Yaskawa INFORM job: BATMAN_ALL2.JBI

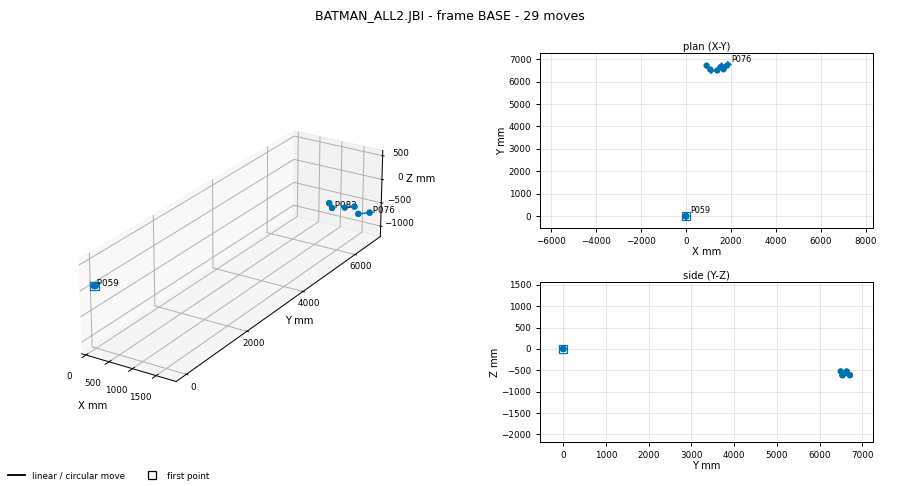
[picture p0: tool path of BATMAN_ALL2.JBI in frame BASE, 29 of 158 moves have a stored position in this frame; points joined in program order, loops and branches not executed]
/JOB
//NAME BATMAN_ALL2
///FOLDERNAME KRIS-SCIANA
//POS
///NPOS 87,87,0,38,0,0
///TOOL 0
///POSTYPE PULSE
///PULSE
C00000=110506,-37041,-50550,-2931,89884,-21361
C00001=114892,-14127,-29600,-10669,91134,-4857
C00002=113309,1036,-13095,-10480,88604,-5183
C00003=113309,1047,-12858,-10479,88468,-5172
C00004=113309,1099,-12019,-10480,87986,-5131
C00005=110003,-19213,-30454,-10104,88460,-6296
C00006=100624,-28655,-35188,-8947,85446,-9259
C00007=100624,-28589,-34530,-8950,85080,-9233
C00008=88503,-50343,-48999,-7293,81608,-13154
C00009=87519,-48373,-46692,-7153,81113,-13463
C00010=87519,-48178,-45668,-7163,80590,-13433
C00011=74941,-63910,-55976,-5229,77890,-17639
C00012=74079,-60203,-53078,-5087,77953,-17939
C00013=74079,-60089,-52614,-5090,77727,-17930
C00014=55396,-72561,-60751,-1908,75512,-24350
C00015=59223,-67103,-56860,-2578,76030,-23030
C00016=59223,-66930,-56247,-2581,75742,-23025
C00017=53352,-67815,-56618,-1545,75365,-25060
C00018=53352,-67667,-56116,-1546,75132,-25057
C00019=64180,-89640,-80007,-3408,78875,-21387
C00020=105889,-74590,-78064,-8027,90261,-8114
C00021=101467,-10036,-27250,4147,89747,-38010
C00022=102269,8905,-7145,5047,92503,-37582
C00023=102269,8938,-6398,5045,92065,-37599
C00024=106927,-8347,-24401,4755,93974,-35953
C00025=117713,-25738,-34686,3963,90797,-32440
C00026=117713,-25680,-33875,3963,90329,-32455
C00027=121342,-12704,-43274,3805,102585,-30865
C00028=122365,-2436,-30975,7466,102876,-21483
C00029=123834,209,-25882,7338,100983,-21103
C00030=123834,88,-25276,7327,100554,-21128
C00031=125992,-4229,-29929,7242,101008,-20372
C00032=126961,-4195,-29168,7180,100477,-20079
C00033=126961,-4277,-28741,7171,100173,-20096
C00034=128213,-6873,-33930,7161,101913,-19574
C00035=136462,-12744,-36389,332,96526,6692
C00036=136057,-12302,-35662,373,96309,6558
C00037=136057,-12373,-35278,373,96036,6558
C00038=138935,-4437,-29695,77,96673,7506
C00039=138935,-4555,-29097,77,96245,7506
C00040=154016,-23376,-48284,-1480,98505,12450
C00041=151429,-25232,-35072,-1194,89379,11690
C00042=149832,-22730,-33163,-1034,89469,11152
C00043=149832,-22673,-32112,-1034,88852,11157
C00044=151805,-20091,-31972,-1235,90121,11807
C00045=159760,14252,-5960,-2031,91919,14440
C00046=159397,21449,3659,-1976,89691,14355
C00047=159397,21501,4652,-1975,89107,14363
C00048=160803,15380,-6921,-2122,93117,14768
C00049=147549,19275,-10198,12019,91012,-52294
C00050=149003,26079,978,11744,87491,-52144
C00051=149003,26016,1819,11745,86950,-52195
C00052=149909,22860,-3198,11576,88263,-51768
C00053=149909,22683,-1380,11579,87076,-51877
C00054=149647,22604,-3622,11626,88432,-51843
C00055=163238,1174,-21239,8981,86572,-47455
C00056=163238,1076,-20285,8983,85943,-47501
C00057=163238,1199,-21452,8978,86716,-47445
C00058=174499,-8738,-29318,6585,85392,-43787
C00059=174499,-8784,-28889,6588,85107,-43802
C00060=175724,-10751,-30896,6317,85233,-43389
C00061=185618,-13733,-32918,4095,84322,-40145
C00062=185618,-13797,-32209,4098,83854,-40160
C00063=192158,-21778,-40833,2582,84794,-37970
C00064=197801,-16179,-34257,1266,83494,-36127
C00065=197801,-16202,-33969,1265,83305,-36129
C00066=201132,-17464,-35697,483,83683,-35023
C00067=201132,-17498,-35315,483,83431,-35024
C00068=201561,-18414,-40963,381,86434,-34873
C00069=152433,-1711,-36929,11228,95909,-50239
C00070=149909,22860,-3198,11576,88263,-51768
C00071=199891,-24183,-46515,806,87858,-35404
C00072=200651,-31220,-49619,-3479,86656,-29192
C00073=201584,-39848,-53424,-8733,85183,-21576
C00074=110806,-28011,-40120,-9545,89205,-14677
C00075=113894,1113,-21993,-10609,94615,-5492
C00076=72814,-67114,-65300,-13368,91768,8253
C00077=115805,-17492,-38928,-13053,98244,-13420
C00078=115343,1086,-18158,-12909,95015,-13235
C00079=116927,-25631,-48082,4098,99115,-32437
C00080=123423,-3162,-32417,7437,103297,-21084
C00081=132585,-17052,-42645,2309,98468,385
C00082=153638,3085,-25046,-14375,106478,-1288
C00083=149417,-20403,-38030,-981,93656,10983
C00084=160973,16174,-17849,-2165,100252,14701
C00085=166397,-29255,-56390,-13219,106573,15875
C00086=18207,-67114,-65300,-13368,91768,8253
BC00000=235494,1186110,777269
BC00001=256125,1186110,671730
BC00002=256125,1186109,671727
BC00003=256125,1186109,671727
BC00004=256125,1186109,671727
BC00005=256125,1186109,671727
BC00006=256125,1186109,671725
BC00007=256125,1186109,671725
BC00008=256125,1186109,671725
BC00009=256125,1186109,671725
BC00010=256125,1186109,671725
BC00011=256125,1186109,671725
BC00012=256125,1186109,671725
BC00013=256125,1186109,671725
BC00014=256125,1186109,671725
BC00015=256125,1186109,671725
BC00016=256125,1186109,671725
BC00017=256125,1186109,671725
BC00018=256125,1186109,671725
BC00019=256125,1186109,671725
BC00020=256125,1186109,671725
BC00021=256125,1186109,671725
BC00022=256125,1186109,671725
BC00023=256125,1186109,671725
BC00024=256125,1186109,671725
BC00025=256125,1186109,671725
BC00026=256125,1186109,671725
BC00027=256125,1186109,671725
BC00028=256125,1186109,671725
BC00029=256125,1186109,671725
BC00030=256125,1186109,671725
BC00031=256125,1186109,671725
BC00032=256125,1186109,671725
BC00033=256125,1186109,671725
BC00034=256125,1186109,671725
BC00035=256125,1186109,671725
BC00036=256125,1186109,671725
BC00037=256125,1186109,671725
BC00038=256125,1186109,671725
BC00039=256125,1186109,671725
BC00040=256125,1186109,671725
BC00041=256125,1186109,671725
BC00042=256125,1186109,671725
BC00043=256125,1186109,671725
BC00044=256125,1186109,671725
BC00045=256125,1186109,671725
BC00046=256124,1186108,671722
BC00047=256124,1186108,671722
BC00048=256124,1186108,671722
BC00049=256125,1186111,610516
BC00050=256125,1186111,610516
BC00051=256125,1186111,610516
BC00052=256125,1186111,610516
BC00053=256125,1186111,610516
BC00054=256125,1186111,610516
BC00055=256125,1186111,610516
BC00056=256125,1186111,610516
BC00057=256125,1186111,610516
BC00058=256125,1186111,610516
BC00059=256125,1186111,610516
BC00060=256125,1186111,610516
BC00061=256125,1186111,610516
BC00062=256125,1186111,610516
BC00063=256125,1186111,610516
BC00064=256125,1186111,610516
BC00065=256125,1186111,610516
BC00066=256125,1186111,610516
BC00067=256125,1186111,610516
BC00068=256125,1186111,610516
BC00069=256125,1186110,610513
BC00070=256125,1186111,610516
BC00071=247912,1186111,610516
BC00072=234351,1186111,753205
BC00073=230913,1186110,814175
BC00074=256125,1186110,753100
BC00075=256125,1186109,671727
BC00076=256125,1186109,671727
BC00077=256125,1186109,671727
BC00078=256125,1186109,671727
BC00079=256125,1186109,671727
BC00080=256125,1186109,671727
BC00081=256125,1186109,671727
BC00082=256125,1186109,671727
BC00083=256125,1186109,671727
BC00084=256125,1186109,671727
BC00085=208948,1186109,671727
BC00086=144067,1278210,991374
///POSTYPE BASE
///RECTAN
///RCONF 0,0,0,0,0,0,0,0,0,0,0,0,0,0,0,0,0,0,0,0,0,0,0,0
P00059=0.483,-0.984,-2.888,0.0000,0.0000,0.0000
P00060=2.327,-2.514,-2.692,0.0000,0.0000,0.0000
P00061=1.575,-3.405,-0.752,0.0000,0.0000,0.0000
P00062=-0.135,-0.848,-1.706,0.0000,0.0000,0.0000
P00063=0.036,-0.654,-3.005,0.0000,0.0000,0.0000
P00064=-0.056,-0.423,-1.596,0.0000,0.0000,0.0000
P00065=-5.731,-1.657,0.588,0.0000,0.0000,0.0000
P00070=0.003,2.805,-1.116,0.0000,0.0000,0.0000
P00071=2.716,0.070,1.352,0.0000,0.0000,0.0000
P00072=1.041,-0.003,-0.797,0.0000,0.0000,0.0000
P00073=-0.961,5.319,-6.157,0.0000,0.0000,0.0000
P00074=1.123,1.944,-5.914,0.0000,0.0000,0.0000
///RCONF 0,1,0,0,0,0,0,0,0,0,0,0,0,0,0,0,0,0,0,0,0,0,0,0
P00075=-1.802,0.025,1.546,0.0000,0.0000,0.0000
///RCONF 0,0,0,0,0,0,0,0,0,0,0,0,0,0,0,0,0,0,0,0,0,0,0,0
P00076=1830.475,6713.589,-615.047,-10.0281,37.5073,-56.2412
P00077=1670.673,6544.317,-616.315,-10.0497,37.5473,-56.2807
P00078=1529.727,6638.522,-525.778,-10.0474,37.5483,-56.2737
P00079=1392.721,6493.935,-525.116,-10.0441,37.5324,-56.2705
P00080=-3.893,-3.240,-0.208,0.0000,0.0000,0.0000
P00081=19.486,11.347,1.262,0.0000,0.0000,0.0000
P00082=1084.422,6532.900,-616.641,-10.0181,37.5185,-126.4483
P00083=916.889,6710.405,-616.123,-10.0077,37.5340,-126.4421
P00098=0.276,2.477,1.230,0.0000,0.0000,0.0000
P00099=-0.837,6.343,-3.499,0.0000,0.0000,0.0000
P00105=-1.846,-0.871,-2.217,0.0000,0.0000,0.0000
P00106=13.000,13.000,-3.000,0.0000,0.0000,0.0000
P00107=-12.000,-8.000,-3.000,0.0000,0.0000,0.0000
P00108=0.000,0.000,-3.000,0.0000,0.0000,0.0000
P00109=4.000,4.000,-1.000,-10.0000,10.0000,-30.0000
P00110=13.000,-10.000,-3.000,0.0000,0.0000,0.0000
P00111=-15.000,15.000,-2.000,0.0000,0.0000,0.0000
P00112=15.000,-7.000,-2.500,0.0000,0.0000,0.0000
P00113=-8.000,10.000,-3.000,0.0000,0.0000,0.0000
P00114=10.000,8.000,-3.000,0.0000,0.0000,0.0000
P00115=-8.000,-11.000,-2.000,0.0000,0.0000,60.0000
P00124=0.000,-50.000,0.000,0.0000,0.0000,0.0000
P00125=0.000,0.000,2.400,0.0000,0.0000,0.0000
P00126=-50.000,0.000,0.000,0.0000,0.0000,0.0000
P00127=50.000,0.000,0.000,0.0000,0.0000,0.0000
//INST
///DATE 2024/07/30 18:50
///COMM NOWY SEARCH
///ATTR SC,RW
///GROUP1 RB1,BS1
NOP
SFTOF
CALL JOB:ONLY_CUT_KM_NEW_SCIANA
MOVJ C00000 BC00000 VJ=15.00
MOVJ C00001 BC00001 VJ=15.00
'POMIAR PRAWA STRONA
MOVL C00002 BC00002 V=250.0
'1
MOVL C00003 BC00003 V=166.7
MOVL C00004 BC00004 V=16.7 PL=0 SRCH RIN#(1)=ON T=1.00 DIS=20.0
TIMER T=0.20
IMOV P125 V=13.3 PL=0
TIMER T=0.20
IMOV P127 V=13.3 PL=0 SRCH RIN#(1)=ON DIS=20.0
TIMER T=0.20
GETS PX070 $PX001
TIMER T=0.10
MOVJ C00005 BC00005 VJ=15.00
'2
MOVL C00006 BC00006 V=50.0
MOVL C00007 BC00007 V=16.7 PL=0 SRCH RIN#(1)=ON T=1.00 DIS=20.0
TIMER T=0.20
IMOV P125 V=13.3 PL=0
TIMER T=0.20
IMOV P127 V=13.3 PL=0 SRCH RIN#(1)=ON DIS=20.0
TIMER T=0.20
GETS PX071 $PX001
TIMER T=0.10
MOVJ C00008 BC00008 VJ=15.00
'3
MOVL C00009 BC00009 V=50.0
MOVL C00010 BC00010 V=16.7 PL=0 SRCH RIN#(1)=ON T=1.00 DIS=20.0
TIMER T=0.20
IMOV P125 V=13.3 PL=0
TIMER T=0.20
IMOV P127 V=13.3 PL=0 SRCH RIN#(1)=ON DIS=20.0
TIMER T=0.20
GETS PX072 $PX001
TIMER T=0.10
MOVJ C00011 BC00011 VJ=15.00
'4
MOVL C00012 BC00012 V=50.0
MOVL C00013 BC00013 V=16.7 PL=0 SRCH RIN#(1)=ON T=1.00 DIS=20.0
TIMER T=0.20
IMOV P125 V=13.3 PL=0
TIMER T=0.20
IMOV P127 V=13.3 PL=0 SRCH RIN#(1)=ON DIS=20.0
TIMER T=0.20
GETS PX073 $PX001
TIMER T=0.10
MOVJ C00014 BC00014 VJ=15.00
'5
MOVL C00015 BC00015 V=50.0
MOVL C00016 BC00016 V=16.7 PL=0 SRCH RIN#(1)=ON T=1.00 DIS=30.0
TIMER T=0.20
IMOV P125 V=13.3 PL=0
TIMER T=0.20
IMOV P127 V=13.3 PL=0 SRCH RIN#(1)=ON DIS=30.0
TIMER T=0.20
GETS PX074 $PX001
TIMER T=0.10
MOVL C00017 BC00017 V=50.0
MOVL C00018 BC00018 V=16.7 PL=0 SRCH RIN#(1)=ON T=1.00 DIS=30.0
TIMER T=0.20
IMOV P125 V=13.3 PL=0
TIMER T=0.20
IMOV P127 V=13.3 PL=0 SRCH RIN#(1)=ON DIS=20.0
TIMER T=0.20
GETS PX075 $PX001
TIMER T=0.10
MOVJ C00019 BC00019 VJ=15.00
MOVJ C00020 BC00020 VJ=30.00
'POMIAR BATMAN
MOVJ C00021 BC00021 VJ=30.00
MOVL C00022 BC00022 V=166.7
MOVL C00023 BC00023 V=13.3 PL=0 SRCH RIN#(1)=ON T=1.00 DIS=20.0
TIMER T=0.20
IMOV P125 V=13.3 PL=0
TIMER T=0.20
IMOV P124 V=13.3 PL=0 SRCH RIN#(1)=ON DIS=20.0
TIMER T=0.20
GETS PX076 $PX001
TIMER T=0.10
MOVJ C00024 BC00024 VJ=30.00
MOVL C00025 BC00025 V=166.7
MOVL C00026 BC00026 V=16.7 PL=0 SRCH RIN#(1)=ON T=1.00 DIS=20.0
TIMER T=0.20
IMOV P125 V=13.3 PL=0
TIMER T=0.20
IMOV P124 V=13.3 PL=0 SRCH RIN#(1)=ON DIS=20.0
TIMER T=0.20
GETS PX077 $PX001
TIMER T=0.10
MOVJ C00027 BC00027 VJ=30.00
MOVJ C00028 BC00028 VJ=30.00
MOVL C00029 BC00029 V=166.7
MOVL C00030 BC00030 V=16.7 PL=0 SRCH RIN#(1)=ON T=1.00 DIS=20.0
TIMER T=0.20
IMOV P125 V=13.3 PL=0
TIMER T=0.20
IMOV P124 V=13.3 PL=0 SRCH RIN#(1)=ON DIS=20.0
TIMER T=0.20
GETS PX078 $PX001
TIMER T=0.10
MOVJ C00031 BC00031 VJ=30.00
MOVL C00032 BC00032 V=166.7
MOVL C00033 BC00033 V=16.7 PL=0 SRCH RIN#(1)=ON T=1.00 DIS=20.0
TIMER T=0.20
IMOV P125 V=13.3 PL=0
TIMER T=0.20
IMOV P124 V=13.3 PL=0 SRCH RIN#(1)=ON DIS=20.0
TIMER T=0.20
GETS PX079 $PX001
TIMER T=0.10
MOVJ C00034 BC00034 VJ=30.00
MOVJ C00035 BC00035 VJ=30.00
MOVL C00036 BC00036 V=166.7
MOVL C00037 BC00037 V=16.7 PL=0 SRCH RIN#(1)=ON T=1.00 DIS=20.0
TIMER T=0.20
IMOV P125 V=13.3 PL=0
TIMER T=0.20
IMOV P124 V=13.3 PL=0 SRCH RIN#(1)=ON DIS=20.0
TIMER T=0.20
GETS PX080 $PX001
TIMER T=0.10
MOVL C00038 BC00038 V=166.7
MOVL C00039 BC00039 V=16.7 PL=0 SRCH RIN#(1)=ON T=1.00 DIS=20.0
TIMER T=0.20
IMOV P125 V=13.3 PL=0
TIMER T=0.20
IMOV P124 V=13.3 PL=0 SRCH RIN#(1)=ON DIS=20.0
TIMER T=0.20
GETS PX081 $PX001
TIMER T=0.10
MOVJ C00040 BC00040 VJ=30.00
MOVJ C00041 BC00041 VJ=30.00
MOVL C00042 BC00042 V=166.7
MOVL C00043 BC00043 V=16.7 PL=0 SRCH RIN#(1)=ON T=1.00 DIS=20.0
TIMER T=0.20
IMOV P125 V=13.3 PL=0
TIMER T=0.20
IMOV P124 V=13.3 PL=0 SRCH RIN#(1)=ON DIS=20.0
TIMER T=0.20
GETS PX082 $PX001
TIMER T=0.10
MOVJ C00044 BC00044 VJ=15.00
MOVJ C00045 BC00045 VJ=30.00
MOVL C00046 BC00046 V=166.7
MOVL C00047 BC00047 V=16.7 PL=0 SRCH RIN#(1)=ON T=1.00 DIS=20.0
TIMER T=0.20
IMOV P125 V=23.0 PL=0
TIMER T=0.20
IMOV P124 V=23.0 PL=0 SRCH RIN#(1)=ON DIS=20.0
TIMER T=0.20
GETS PX083 $PX001
TIMER T=0.10
MOVJ C00048 BC00048 VJ=30.00
'KONIEC POMIAR BATMAN 1STR
SFTOF
MOVJ C00049 BC00049 VJ=15.00
'1
MOVL C00050 BC00050 V=166.7
MOVL C00051 BC00051 V=16.7 PL=0 SRCH RIN#(1)=ON T=1.00 DIS=20.0
TIMER T=0.20
IMOV P125 V=13.3 PL=0
TIMER T=0.20
IMOV P126 V=13.3 PL=0 SRCH RIN#(1)=ON DIS=20.0
TIMER T=0.20
GETS PX059 $PX001
TIMER T=0.10
MOVL C00052 BC00052 V=166.7
MOVL C00053 BC00053 V=16.7 PL=0 SRCH RIN#(1)=ON T=1.00 DIS=20.0
TIMER T=0.20
IMOV P125 V=13.3 PL=0
TIMER T=0.20
IMOV P126 V=13.3 PL=0 SRCH RIN#(1)=ON DIS=20.0
TIMER T=0.20
GETS PX060 $PX001
TIMER T=0.10
MOVJ C00054 BC00054 VJ=0.78
'2
MOVL C00055 BC00055 V=50.0
MOVL C00056 BC00056 V=16.7 PL=0 SRCH RIN#(1)=ON T=1.00 DIS=20.0
TIMER T=0.20
IMOV P125 V=13.3 PL=0
TIMER T=0.20
IMOV P126 V=13.3 PL=0 SRCH RIN#(1)=ON DIS=20.0
TIMER T=0.20
GETS PX061 $PX001
TIMER T=0.10
MOVJ C00057 BC00057 VJ=0.78
'3
MOVL C00058 BC00058 V=50.0
MOVL C00059 BC00059 V=16.7 PL=0 SRCH RIN#(1)=ON T=1.00 DIS=20.0
TIMER T=0.20
IMOV P125 V=13.3 PL=0
TIMER T=0.20
IMOV P126 V=13.3 PL=0 SRCH RIN#(1)=ON DIS=20.0
TIMER T=0.20
GETS PX062 $PX001
TIMER T=0.10
MOVJ C00060 BC00060 VJ=0.78
'4
MOVL C00061 BC00061 V=50.0
MOVL C00062 BC00062 V=16.7 PL=0 SRCH RIN#(1)=ON T=1.00 DIS=20.0
TIMER T=0.20
IMOV P125 V=13.3 PL=0
TIMER T=0.20
IMOV P126 V=13.3 PL=0 SRCH RIN#(1)=ON DIS=20.0
TIMER T=0.20
GETS PX063 $PX001
TIMER T=0.10
MOVJ C00063 BC00063 VJ=30.00
'5
MOVL C00064 BC00064 V=50.0
MOVL C00065 BC00065 V=16.7 PL=0 SRCH RIN#(1)=ON T=1.00 DIS=20.0
TIMER T=0.20
IMOV P125 V=13.3 PL=0
TIMER T=0.20
IMOV P126 V=13.3 PL=0 SRCH RIN#(1)=ON DIS=20.0
TIMER T=0.20
GETS PX064 $PX001
TIMER T=0.10
MOVL C00066 BC00066 V=50.0
MOVL C00067 BC00067 V=16.7 PL=0 SRCH RIN#(1)=ON T=1.00 DIS=20.0
TIMER T=0.20
IMOV P125 V=13.3 PL=0
TIMER T=0.20
IMOV P126 V=13.3 PL=0 SRCH RIN#(1)=ON DIS=20.0
TIMER T=0.20
GETS PX065 $PX001
TIMER T=0.10
MOVJ C00068 BC00068 VJ=15.00
'********
'********
'********
MOVJ C00069 BC00069 VJ=15.00
MOVL C00070 BC00070 V=333.3
MACRO1 MJ#(0) ARGF7
SFTOF
SFTON P109
MOVL P059 V=83.3
ARCON
SFTOF
SFTON P099
MOVL P060 V=10.8
MOVL P061 V=10.8
MOVL P062 V=10.8
MOVL P063 V=10.8
MOVL P064 V=10.8
MOVL P065 V=10.8
ARCOF
MOVJ C00071 BC00071 VJ=15.00
SFTOF
MOVJ C00072 BC00072 VJ=50.00
MOVJ C00073 BC00073 VJ=15.00
MOVJ C00074 BC00074 VJ=15.00
SFTON P115
MOVJ C00075 BC00075 VJ=15.00
MOVL P070 V=83.3
ARCON
SFTOF
SFTON P098
MOVL P071 V=10.8
MOVL P072 V=10.8
MOVL P073 V=10.8
MOVL P074 V=10.8
MOVL P075 V=10.8
ARCOF
SFTOF
MOVJ C00076 BC00076 VJ=15.00
MOVJ C00077 BC00077 VJ=30.00
MOVJ C00078 BC00078 VJ=30.00
SFTON P110
MOVL P076 V=83.3
SFTOF
ARCON
SFTON P108
MOVL P076 V=10.8
MOVL P077 V=10.8
SFTON P111
MOVL P077 V=10.8
ARCOF
SFTOF
MOVJ C00079 BC00079 VJ=30.00
MOVJ C00080 BC00080 VJ=30.00
SFTON P112
MOVL P078 V=83.3
ARCON
SFTOF
SFTON P108
MOVL P078 V=10.8
MOVL P079 V=10.8
SFTOF
SFTON P113
MOVL P079 V=10.8
ARCOF
SFTOF
MOVJ C00081 BC00081 VJ=30.00
SFTON P114
MOVL P080 V=83.3
SFTOF
ARCON
SFTON P108
MOVL P080 V=10.8
MOVL P081 V=10.8
SFTOF
SFTON P105
MOVL P081 V=10.8
SFTOF
ARCOF
MOVJ C00082 BC00082 VJ=30.00
MOVJ C00083 BC00083 VJ=30.00
SFTON P106
MOVL P082 V=83.3
SFTOF
ARCON
SFTON P108
MOVL P082 V=10.8
MOVL P083 V=10.8
SFTOF
SFTON P107
MOVL P083 V=10.8
SFTOF
ARCOF
MOVJ C00084 BC00084 VJ=30.00
MOVJ C00085 BC00085 VJ=30.00
MOVJ C00086 BC00086 VJ=80.00
CALL JOB:ONLY_CUT_KM_NEW_SCIANA
END
